Staubli VAL3: saveCycle.pjx

--- saveCycle.pjx ---
Parameters version=s7.2.1 stackSize=5000 millimeterUnit=true
Data file=saveCycle.dtx

--- saveCycle.dtx ---
public bool bLoop = true
public num nDoneCycle
public num nDoneEnd
public num nDoneStart
public num nTime
public num nTotalCycle
public num nTotalEnd
public num nTotalStart = 1
public num nType = 1
public string sLoadEnd
public string sLoadProg
public string sLoadStart
